PROGRAM Messages
VAR

END_VAR

sMessages:='System Ok';


IF EmergencyStop_Latch THEN
	sMessages:='EMERGENCY  STOP!';
END_IF

END_PROGRAM

(* stored: Version 1.1.0.1, ProductVersion 3.1.4024.15
   POU Messages: Id {4986c3eb-32c8-45f8-942f-4b1897b9fd51}, SpecialFunc None *)
